// TIA Portal V19 export
TYPE "C403_STU_LVE_TYPIC"
   STRUCT
      LCK_STOP { ExternalAccessible := 'False'; ExternalVisible := 'False'; ExternalWritable := 'False'} : Array[1..7, 0..40] of Int;   // Lijst van detectiepunten die een stilstand signaleren
      LCK_SOS { ExternalAccessible := 'False'; ExternalVisible := 'False'; ExternalWritable := 'False'} : Array[1..7, 0..40] of Int;   // Lijst van detectiepunten die een snelheidsonderschrijding signaleren
      LCK_NEG { ExternalAccessible := 'False'; ExternalVisible := 'False'; ExternalWritable := 'False'} : USInt;   // Ja = Spookrijder detectie vergrendeld (niet actief)
   END_STRUCT;
END_TYPE
